FUNCTION_BLOCK FB_EthercatMaster
VAR_INPUT
    NetId 						AT %I*:	T_AmsNetIdArr;
END_VAR
VAR_OUTPUT
END_VAR
VAR
	sNetId:						T_AmsNetID;
	fbGetMasterState: 			FB_EcGetMasterDevState;
	fbGetSlaveCount: 			FB_EcGetSlaveCount;
END_VAR

IF sNetId = '' THEN
	sNetId:= F_CreateAmsNetId(NetId);
	fbGetMasterState.sNetId:= sNetId;
END_IF

fbGetMasterState(sNetId:= sNetId);

fbGetSlaveCount(sNetId:= sNetId);

END_FUNCTION_BLOCK

(* stored: Version 1.1.0.1
   POU FB_EthercatMaster: Id {8d40e3a5-69ef-036b-1c31-1dbf1ede6c85}, SpecialFunc None *)
